{attribute 'GeneratedUsingTerminal: EP1312-0001-0016'}
{attribute addProperty BoxType "EP1312-0001-0016"}
{attribute addProperty Id "A_0038_EP1518_0002_0016EP1518_1B7BBD8659A_0039_EP1518_0002_0017EP1518_1B7BBD8659A_0040_EP1518_0002_0018EP1518_1B7BBD8659A_0041_EP1518_0002_0019EP1518_1B7BBD8659A_0042_EP1809_0021_0016EP1809_FD7895E220A_0043_EP1809_0021_0017EP1809_FD7895E220A_0044_EP1809_0022_0017EP1809_FD7895E220A_0045_EP1809_0022_0018EP1809_FD7895E220A_0046_EP1809_0042_0018EP1809_96022ACE20A_0047_EP1809_0042_0019EP1809_6EEA635020A_0048_EP1816_0003_0016EP1816_9F97CFEF32A_0049_EP1816_0008_0016EP1816_6F7ED0EC30A_0050_EP1816_0008_0017EP1816_6F7ED0EC30A_0051_EP1816_0008_0018EP1816_6247929530A_0052_EP1816_0008_0019EP1816_6247929530A_0053_EP1816_0008_0020EP1816_6247929530A_0054_EP1816_1008_0016EP1816_12F8118132A_0055_EP1816_1008_0017EP1816_12F8118132A_0056_EP1816_3008_0016EP1816_4FA00BC356A_0057_EP1816_3008_0017EP1816_4FA00BC356A_0058_EP1816_3008_0018EP1816_4FA00BC356A_0059_EP1819_0021_0016EP1819_FD7895E220A_0060_EP1819_0021_0017EP1819_FD7895E220A_0061_EP1819_0022_0016EP1819_FD7895E220A_0062_EP1819_0022_0017EP1819_FD7895E220A_0063_EP1859_0042_0018EP1859_8B8263DA20A_0064_EP1859_0042_0019EP1859_592B0CC320"}
{attribute addProperty CRC "2764110689"}
{attribute addProperty Size "890"}
TYPE A_0037_EP1312_0001_0016_A4C0FB61 EXTENDS EP1312_AB5A9467 :
STRUCT
	{attribute addProperty Name "A_0038_EP1518_0002_0016"}
	A_0038_EP1518_0002_0016 : EP1518_1B7BBD86;
	{attribute addProperty Name "A_0039_EP1518_0002_0017"}
	A_0039_EP1518_0002_0017 : EP1518_1B7BBD86;
	{attribute addProperty Name "A_0040_EP1518_0002_0018"}
	A_0040_EP1518_0002_0018 : EP1518_1B7BBD86;
	{attribute addProperty Name "A_0041_EP1518_0002_0019"}
	A_0041_EP1518_0002_0019 : EP1518_1B7BBD86;
	{attribute addProperty Name "A_0042_EP1809_0021_0016"}
	A_0042_EP1809_0021_0016 : EP1809_FD7895E2;
	{attribute addProperty Name "A_0043_EP1809_0021_0017"}
	A_0043_EP1809_0021_0017 : EP1809_FD7895E2;
	{attribute addProperty Name "A_0044_EP1809_0022_0017"}
	A_0044_EP1809_0022_0017 : EP1809_FD7895E2;
	{attribute addProperty Name "A_0045_EP1809_0022_0018"}
	A_0045_EP1809_0022_0018 : EP1809_FD7895E2;
	{attribute addProperty Name "A_0046_EP1809_0042_0018"}
	A_0046_EP1809_0042_0018 : EP1809_96022ACE;
	{attribute addProperty Name "A_0047_EP1809_0042_0019"}
	A_0047_EP1809_0042_0019 : EP1809_6EEA6350;
	{attribute addProperty Name "A_0048_EP1816_0003_0016"}
	A_0048_EP1816_0003_0016 : EP1816_9F97CFEF;
	{attribute addProperty Name "A_0049_EP1816_0008_0016"}
	A_0049_EP1816_0008_0016 : EP1816_6F7ED0EC;
	{attribute addProperty Name "A_0050_EP1816_0008_0017"}
	A_0050_EP1816_0008_0017 : EP1816_6F7ED0EC;
	{attribute addProperty Name "A_0051_EP1816_0008_0018"}
	A_0051_EP1816_0008_0018 : EP1816_62479295;
	{attribute addProperty Name "A_0052_EP1816_0008_0019"}
	A_0052_EP1816_0008_0019 : EP1816_62479295;
	{attribute addProperty Name "A_0053_EP1816_0008_0020"}
	A_0053_EP1816_0008_0020 : EP1816_62479295;
	{attribute addProperty Name "A_0054_EP1816_1008_0016"}
	A_0054_EP1816_1008_0016 : EP1816_12F81181;
	{attribute addProperty Name "A_0055_EP1816_1008_0017"}
	A_0055_EP1816_1008_0017 : EP1816_12F81181;
	{attribute addProperty Name "A_0056_EP1816_3008_0016"}
	A_0056_EP1816_3008_0016 : EP1816_4FA00BC3;
	{attribute addProperty Name "A_0057_EP1816_3008_0017"}
	A_0057_EP1816_3008_0017 : EP1816_4FA00BC3;
	{attribute addProperty Name "A_0058_EP1816_3008_0018"}
	A_0058_EP1816_3008_0018 : EP1816_4FA00BC3;
	{attribute addProperty Name "A_0059_EP1819_0021_0016"}
	A_0059_EP1819_0021_0016 : EP1819_FD7895E2;
	{attribute addProperty Name "A_0060_EP1819_0021_0017"}
	A_0060_EP1819_0021_0017 : EP1819_FD7895E2;
	{attribute addProperty Name "A_0061_EP1819_0022_0016"}
	A_0061_EP1819_0022_0016 : EP1819_FD7895E2;
	{attribute addProperty Name "A_0062_EP1819_0022_0017"}
	A_0062_EP1819_0022_0017 : EP1819_FD7895E2;
	{attribute addProperty Name "A_0063_EP1859_0042_0018"}
	A_0063_EP1859_0042_0018 : EP1859_8B8263DA;
	{attribute addProperty Name "A_0064_EP1859_0042_0019"}
	A_0064_EP1859_0042_0019 : EP1859_592B0CC3;
END_STRUCT
END_TYPE

(* stored: Version 1.2.0.0, ProductVersion 3.1.4024.9
   DUT A_0037_EP1312_0001_0016_A4C0FB61: Id {5ec2245e-ffb2-42ce-b9a0-41f17662a8a9} *)
